FUNCTION_BLOCK TAdsWriteBySymbolName
VAR
    Execution : TExecution;
    StateMonitor : TValueMonitor;
    State : INT;

	AmsNetId            : T_AmsNetId;
	Port                : T_AmsPort;
	SymbolName          : STRING;
    WriteDataAddress    : PVOID;
    WriteDataLength     : UDINT;    
    KeepSymbolHandle    : BOOL;  
	SymbolHandle 	    : DWORD := 0;
    RetryCounter : TCounter;

    AdsReadWrite_GetSymHandle : TAdsReadWrite;
    AdsWrite_WriteToSymbol    : TAdsWrite;
    AdsWrite_ReleaseSymHandle : TAdsWrite;
END_VAR
VAR CONSTANT
    sInit          : INT := 0;
    sGetHandle     : INT := 1;
    sWriteData     : INT := 2;
    sReleaseHandle : INT := 3;
END_VAR

StateMonitor.Test(State);
CASE State OF
    sInit:
        IF Execution.Starting THEN
            Execution.SetBusy();
            RetryCounter.Reset();
            IF SymbolHandle = 0 THEN
                State := sGetHandle;
            ELSE
                State := sWriteData;
            END_IF
		END_IF
        
    sGetHandle: 
        IF StateMonitor.Changed THEN
            // Get a symbol handle from the runtime...
            AdsReadWrite_GetSymHandle.Execute(
                AmsNetId            := AmsNetId, 
                Port                := Port, 
                IndexGroup          := ADSIGRP_SYM_HNDBYNAME, 
                IndexOffset         := 0, 
                ArgsAddress         := ADR(SymbolName), 
                ArgsLength          := INT_TO_UDINT(LEN(SymbolName)), 
                ReturnValueAddress  := ADR(SymbolHandle), 
                ReturnValueLength   := SIZEOF(SymbolHandle));
        ELSE
            IF AdsReadWrite_GetSymHandle.ExecutionResult.Done THEN
                State := sWriteData;
			END_IF
            IF AdsReadWrite_GetSymHandle.ExecutionResult.Error THEN
                Execution.SetError(AdsReadWrite_GetSymHandle.ExecutionResult.ErrorId);
                SymbolHandle := 0;
                State := sInit;
			END_IF
        END_IF
        
    sWriteData: 
        IF StateMonitor.Changed THEN
            // Write the data to the symbol...
            AdsWrite_WriteToSymbol.Execute(
                AmsNetId        := AmsNetId, 
                Port            := Port, 
                IndexGroup      := ADSIGRP_SYM_VALBYHND, 
                IndexOffset     := SymbolHandle, 
                DataLength      := WriteDataLength, 
                DataAddress     := WriteDataAddress);
        ELSE
            IF AdsWrite_WriteToSymbol.ExecutionResult.Done THEN
                IF KeepSymbolHandle THEN
                    Execution.SetDone();
                    State := sInit;
                ELSE
                    State := sReleaseHandle;
				END_IF
                
            ELSIF AdsWrite_WriteToSymbol.ExecutionResult.Error THEN
                // Detect if it failed due to an online change invalidating the symbol handle...
                IF 
                    AdsWrite_WriteToSymbol.ExecutionResult.ErrorId = E_AdsErr.DEVICE_SYMBOLVERSIONINVALID 
                 OR
                    AdsWrite_WriteToSymbol.ExecutionResult.ErrorId = E_AdsErr.DEVICE_SYMBOLNOTACTIVE 
                THEN
                    IF RetryCounter.Value > 0 THEN
                        Execution.SetError(AdsWrite_WriteToSymbol.ExecutionResult.ErrorId);
                        SymbolHandle := 0;
                        State := sInit;
                    ELSE
                        RetryCounter.Inc();
                        SymbolHandle := 0;
                        State := sGetHandle;
                    END_IF
                ELSE
                    State := sReleaseHandle;
				END_IF
			END_IF
		END_IF

    sReleaseHandle:    
        IF StateMonitor.Changed THEN
            // Release the symbol handle......
            AdsWrite_ReleaseSymHandle.Execute(
                AmsNetId        := AmsNetId, 
                Port            := Port, 
                IndexGroup      := ADSIGRP_SYM_RELEASEHND, 
                IndexOffset     := SymbolHandle, 
                DataLength      := 0, 
                DataAddress     := 0);
        ELSE
            IF AdsWrite_ReleaseSymHandle.ExecutionResult.Done THEN
                // Handle write error to the symbol...
                IF AdsWrite_WriteToSymbol.ExecutionResult.Error THEN
                    Execution.SetError(AdsWrite_WriteToSymbol.ExecutionResult.ErrorId);
                ELSE
                    Execution.SetDone();
				END_IF
                SymbolHandle := 0;
                State := sInit;
            ELSIF AdsWrite_ReleaseSymHandle.ExecutionResult.Error THEN
                // Handle release handle error...
                Execution.SetError(AdsWrite_ReleaseSymHandle.ExecutionResult.ErrorId);
                SymbolHandle := 0;
                State := sInit;
            ELSIF AdsWrite_WriteToSymbol.ExecutionResult.Error THEN
                // Handle Write To Symbol error...
                Execution.SetError(AdsWrite_WriteToSymbol.ExecutionResult.ErrorId);
                SymbolHandle := 0;
                State := sInit;
			END_IF
		END_IF

END_CASE

AdsReadWrite_GetSymHandle();
AdsWrite_WriteToSymbol();
AdsWrite_ReleaseSymHandle();

METHOD Execute : BOOL
VAR_INPUT
	AmsNetId            : T_AmsNetId;
	Port                : T_AmsPort;
	SymbolName          : STRING;
    WriteDataAddress    : PVOID;
    WriteDataLength     : UDINT;  
    KeepSymbolHandle    : BOOL;  
END_VAR
THIS^.AmsNetId          := AmsNetId;
THIS^.Port              := Port;
THIS^.SymbolName        := SymbolName;
THIS^.WriteDataAddress  := WriteDataAddress;
THIS^.WriteDataLength   := WriteDataLength;
THIS^.KeepSymbolHandle  := KeepSymbolHandle;

Execute := Execution.Start();
END_METHOD

PROPERTY ExecutionResult : IExecutionResult
GET
ExecutionResult := Execution;
END_GET
END_PROPERTY

END_FUNCTION_BLOCK

(* stored: Version 1.1.0.1, ProductVersion 3.1.4024.3
   POU TAdsWriteBySymbolName: Id {53082c2a-90eb-4e71-93b4-409c3d4e3399}, SpecialFunc None
   Method Execute: Id {dd0b3e87-79eb-4d2d-a0af-07cbd2daf4e4}
   Property ExecutionResult: Id {0ea02708-d4b6-0176-35a7-d44968e802a6}
   Get Get: Id {58100c02-dcb0-03e6-2857-2a6e914e8fd4} *)
